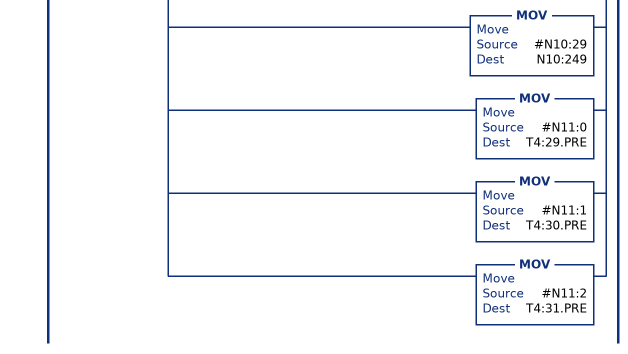
% Rung: 0 %
SOR SBR BST SUB N10:253 1 N10:254 NXB MUL N10:254 30 S:24 NXB MOV #N10:0 T4:0.PRE NXB MOV #N10:1 T4:1.PRE NXB MOV #N10:2 T4:2.PRE NXB MOV #N10:3 T4:3.PRE NXB MOV #N10:4 T4:4.PRE NXB MOV #N10:5 T4:5.PRE NXB MOV #N10:6 T4:6.PRE NXB MOV #N10:7 T4:7.PRE NXB MOV #N10:8 T4:8.PRE NXB MOV #N10:9 T4:9.PRE NXB MOV #N10:10 T4:11.PRE NXB MOV #N10:11 T4:12.PRE NXB MOV #N10:12 T4:13.PRE NXB MOV #N10:13 T4:15.PRE NXB MOV #N10:14 T4:18.PRE NXB MOV #N10:15 T4:19.PRE NXB MOV #N10:16 T4:20.PRE NXB MOV #N10:17 T4:21.PRE NXB MOV #N10:18 T4:22.PRE NXB MOV #N10:19 T4:25.PRE NXB MOV #N10:20 N10:240 NXB MOV #N10:21 N10:241 NXB MOV #N10:22 N10:242 NXB MOV #N10:23 N10:243 NXB MOV #N10:24 N10:244 NXB MOV #N10:25 N10:245 NXB MOV #N10:26 N10:246 NXB MOV #N10:27 N10:247 NXB MOV #N10:28 N10:248 NXB MOV #N10:29 N10:249 NXB MOV #N11:0 T4:29.PRE NXB MOV #N11:1 T4:30.PRE NXB MOV #N11:2 T4:31.PRE BND EOR
%   S:24  "Index Register" %

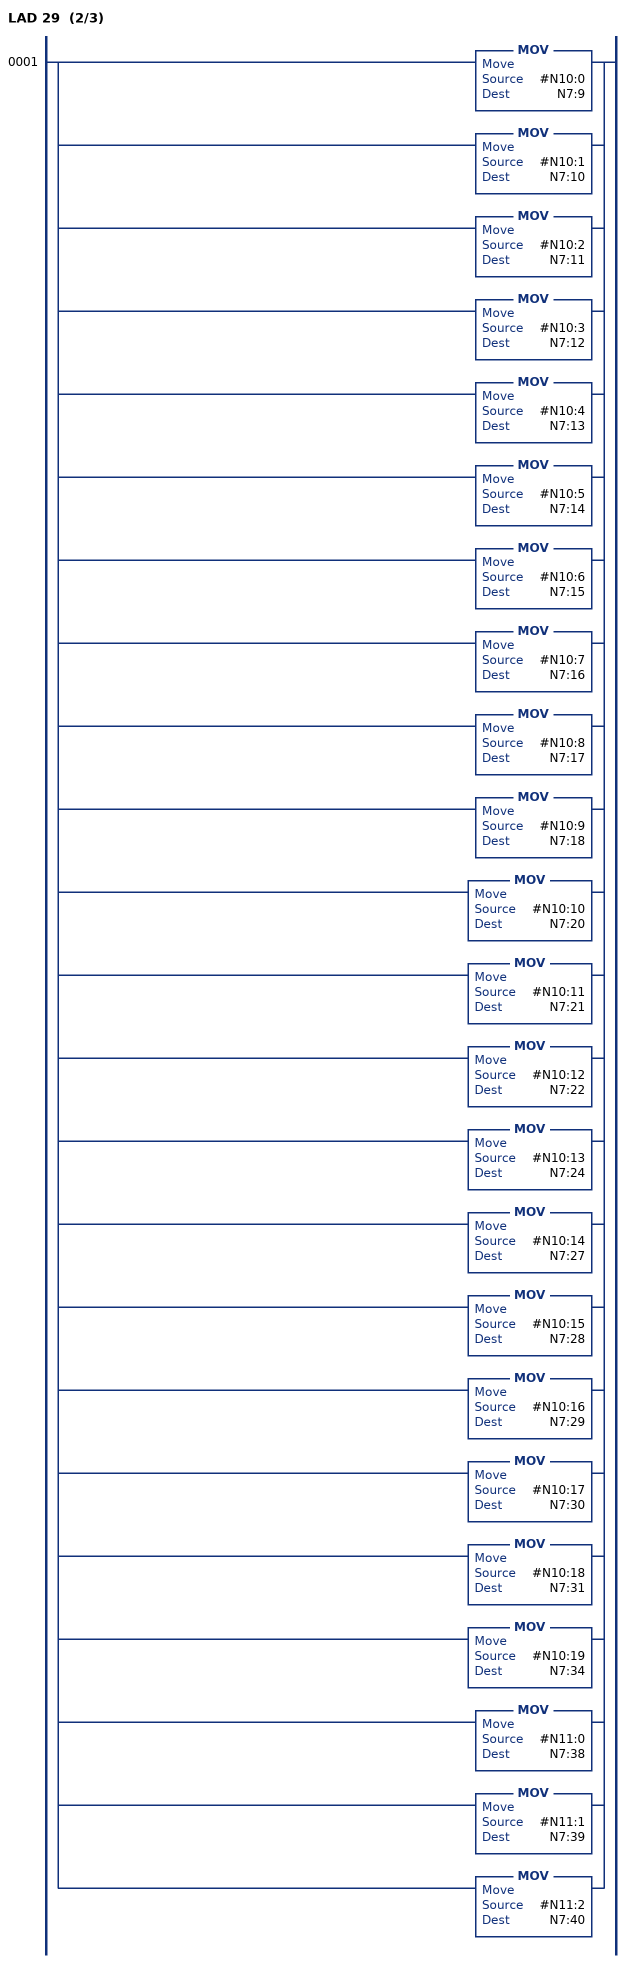
% Rung: 1 %
SOR BST MOV #N10:0 N7:9 NXB MOV #N10:1 N7:10 NXB MOV #N10:2 N7:11 NXB MOV #N10:3 N7:12 NXB MOV #N10:4 N7:13 NXB MOV #N10:5 N7:14 NXB MOV #N10:6 N7:15 NXB MOV #N10:7 N7:16 NXB MOV #N10:8 N7:17 NXB MOV #N10:9 N7:18 NXB MOV #N10:10 N7:20 NXB MOV #N10:11 N7:21 NXB MOV #N10:12 N7:22 NXB MOV #N10:13 N7:24 NXB MOV #N10:14 N7:27 NXB MOV #N10:15 N7:28 NXB MOV #N10:16 N7:29 NXB MOV #N10:17 N7:30 NXB MOV #N10:18 N7:31 NXB MOV #N10:19 N7:34 NXB MOV #N11:0 N7:38 NXB MOV #N11:1 N7:39 NXB MOV #N11:2 N7:40 BND EOR

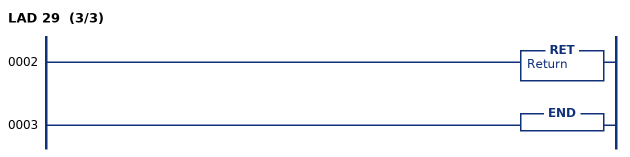
% Rung: 2 %
SOR RET EOR
% Rung: 3 %
SOR END EOR

LADDER 30
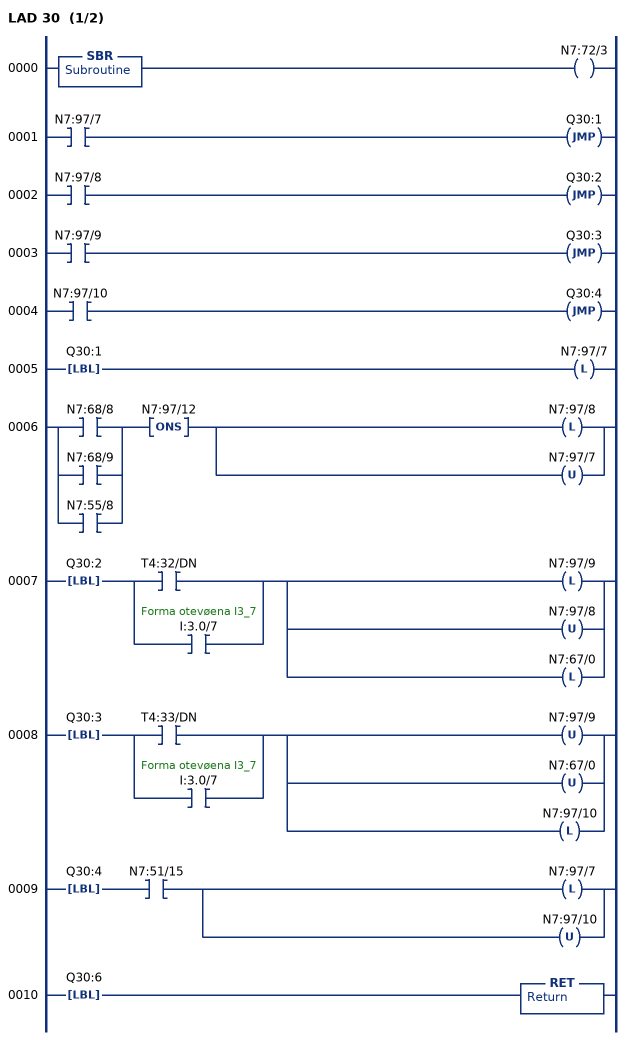
% Rung: 0 %
SOR SBR OTE N7:72/3 EOR
% Rung: 1 %
SOR XIC N7:97/7 JMP Q30:1 EOR
% Rung: 2 %
SOR XIC N7:97/8 JMP Q30:2 EOR
% Rung: 3 %
SOR XIC N7:97/9 JMP Q30:3 EOR
% Rung: 4 %
SOR XIC N7:97/10 JMP Q30:4 EOR
% Rung: 5 %
SOR LBL Q30:1 OTL N7:97/7 EOR
% Rung: 6 %
SOR BST XIC N7:68/8 NXB BST XIC N7:68/9 NXB XIC N7:55/8 BND BND OSR N7:97/12 BST OTL N7:97/8 NXB OTU N7:97/7 BND EOR
% Rung: 7 %
SOR LBL Q30:2 BST XIC T4:32/DN NXB XIC I:3.0/7 BND BST OTL N7:97/9 NXB BST OTU N7:97/8 NXB OTL N7:67/0 BND BND EOR
%   I:3.0/7  I3_7  "Forma otevøena" %
% Rung: 8 %
SOR LBL Q30:3 BST XIC T4:33/DN NXB XIC I:3.0/7 BND BST OTU N7:97/9 NXB BST OTU N7:67/0 NXB OTL N7:97/10 BND BND EOR
%   I:3.0/7  I3_7  "Forma otevøena" %
% Rung: 9 %
SOR LBL Q30:4 XIC N7:51/15 BST OTL N7:97/7 NXB OTU N7:97/10 BND EOR
% Rung: 10 %
SOR LBL Q30:6 RET EOR

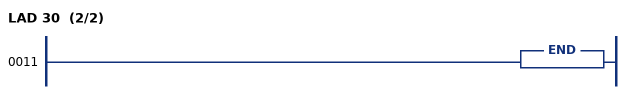
% Rung: 11 %
SOR END EOR

LADDER 31
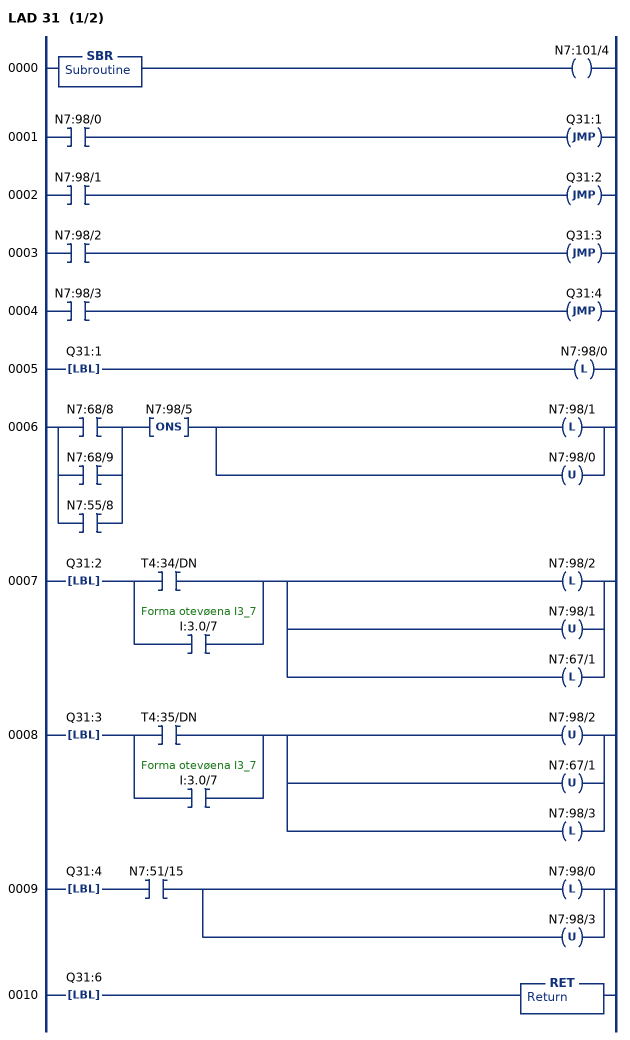
% Rung: 0 %
SOR SBR OTE N7:101/4 EOR
% Rung: 1 %
SOR XIC N7:98/0 JMP Q31:1 EOR
% Rung: 2 %
SOR XIC N7:98/1 JMP Q31:2 EOR
% Rung: 3 %
SOR XIC N7:98/2 JMP Q31:3 EOR
% Rung: 4 %
SOR XIC N7:98/3 JMP Q31:4 EOR
% Rung: 5 %
SOR LBL Q31:1 OTL N7:98/0 EOR
% Rung: 6 %
SOR BST XIC N7:68/8 NXB BST XIC N7:68/9 NXB XIC N7:55/8 BND BND OSR N7:98/5 BST OTL N7:98/1 NXB OTU N7:98/0 BND EOR
% Rung: 7 %
SOR LBL Q31:2 BST XIC T4:34/DN NXB XIC I:3.0/7 BND BST OTL N7:98/2 NXB BST OTU N7:98/1 NXB OTL N7:67/1 BND BND EOR
%   I:3.0/7  I3_7  "Forma otevøena" %
% Rung: 8 %
SOR LBL Q31:3 BST XIC T4:35/DN NXB XIC I:3.0/7 BND BST OTU N7:98/2 NXB BST OTU N7:67/1 NXB OTL N7:98/3 BND BND EOR
%   I:3.0/7  I3_7  "Forma otevøena" %
% Rung: 9 %
SOR LBL Q31:4 XIC N7:51/15 BST OTL N7:98/0 NXB OTU N7:98/3 BND EOR
% Rung: 10 %
SOR LBL Q31:6 RET EOR

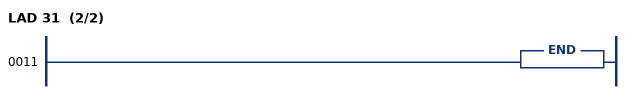
% Rung: 11 %
SOR END EOR

LADDER 32
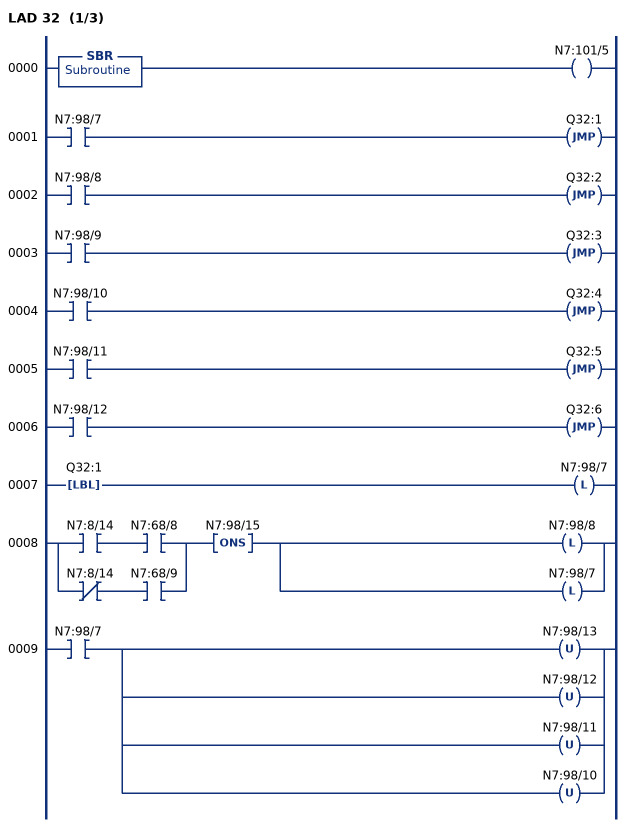
% Rung: 0 %
SOR SBR OTE N7:101/5 EOR
% Rung: 1 %
SOR XIC N7:98/7 JMP Q32:1 EOR
% Rung: 2 %
SOR XIC N7:98/8 JMP Q32:2 EOR
% Rung: 3 %
SOR XIC N7:98/9 JMP Q32:3 EOR
% Rung: 4 %
SOR XIC N7:98/10 JMP Q32:4 EOR
% Rung: 5 %
SOR XIC N7:98/11 JMP Q32:5 EOR
% Rung: 6 %
SOR XIC N7:98/12 JMP Q32:6 EOR
% Rung: 7 %
SOR LBL Q32:1 OTL N7:98/7 EOR
% Rung: 8 %
SOR BST XIC N7:8/14 XIC N7:68/8 NXB XIO N7:8/14 XIC N7:68/9 BND OSR N7:98/15 BST OTL N7:98/8 NXB OTL N7:98/7 BND EOR
% Rung: 9 %
SOR XIC N7:98/7 BST OTU N7:98/13 NXB BST OTU N7:98/12 NXB BST OTU N7:98/11 NXB OTU N7:98/10 BND BND BND EOR

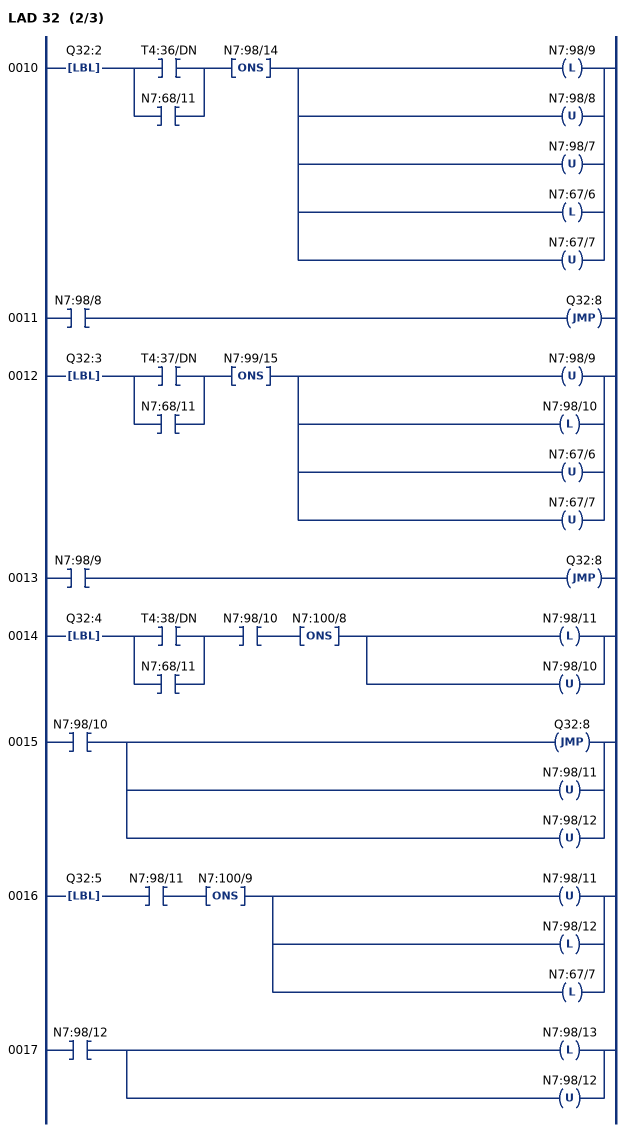
% Rung: 10 %
SOR LBL Q32:2 BST XIC T4:36/DN NXB XIC N7:68/11 BND OSR N7:98/14 BST OTL N7:98/9 NXB BST BST OTU N7:98/8 NXB OTU N7:98/7 BND NXB BST OTL N7:67/6 NXB OTU N7:67/7 BND BND BND EOR
% Rung: 11 %
SOR XIC N7:98/8 JMP Q32:8 EOR
% Rung: 12 %
SOR LBL Q32:3 BST XIC T4:37/DN NXB XIC N7:68/11 BND OSR N7:99/15 BST OTU N7:98/9 NXB BST OTL N7:98/10 NXB BST OTU N7:67/6 NXB OTU N7:67/7 BND BND BND EOR
% Rung: 13 %
SOR XIC N7:98/9 JMP Q32:8 EOR
% Rung: 14 %
SOR LBL Q32:4 BST XIC T4:38/DN NXB XIC N7:68/11 BND XIC N7:98/10 OSR N7:100/8 BST OTL N7:98/11 NXB OTU N7:98/10 BND EOR
% Rung: 15 %
SOR XIC N7:98/10 BST JMP Q32:8 NXB BST OTU N7:98/11 NXB OTU N7:98/12 BND BND EOR
% Rung: 16 %
SOR LBL Q32:5 XIC N7:98/11 OSR N7:100/9 BST BST OTU N7:98/11 NXB OTL N7:98/12 BND NXB OTL N7:67/7 BND EOR
% Rung: 17 %
SOR XIC N7:98/12 BST OTL N7:98/13 NXB OTU N7:98/12 BND EOR

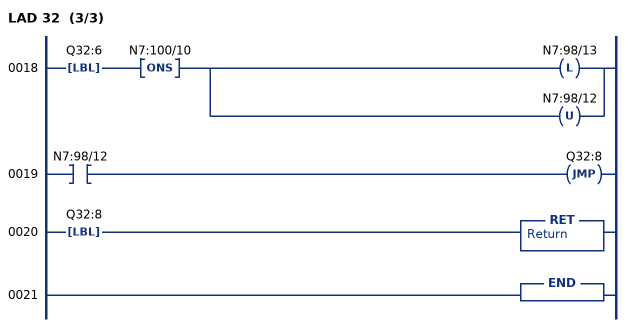
% Rung: 18 %
SOR LBL Q32:6 OSR N7:100/10 BST OTL N7:98/13 NXB OTU N7:98/12 BND EOR
% Rung: 19 %
SOR XIC N7:98/12 JMP Q32:8 EOR
% Rung: 20 %
SOR LBL Q32:8 RET EOR
% Rung: 21 %
SOR END EOR

LADDER 33
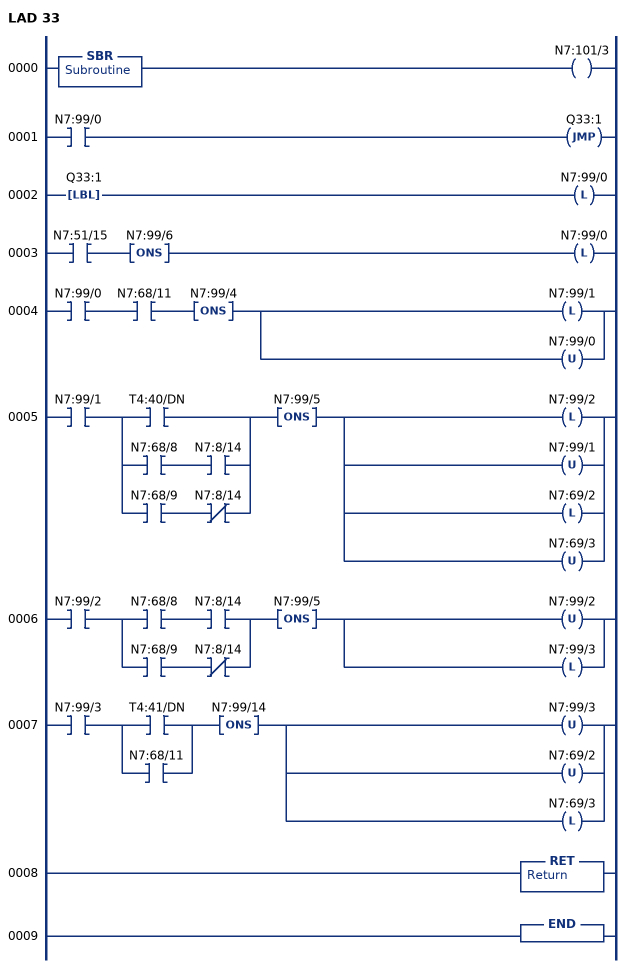
% Rung: 0 %
SOR SBR OTE N7:101/3 EOR
% Rung: 1 %
SOR XIC N7:99/0 JMP Q33:1 EOR
% Rung: 2 %
SOR LBL Q33:1 OTL N7:99/0 EOR
% Rung: 3 %
SOR XIC N7:51/15 OSR N7:99/6 OTL N7:99/0 EOR
% Rung: 4 %
SOR XIC N7:99/0 XIC N7:68/11 OSR N7:99/4 BST OTL N7:99/1 NXB OTU N7:99/0 BND EOR
% Rung: 5 %
SOR XIC N7:99/1 BST XIC T4:40/DN NXB BST XIC N7:68/8 XIC N7:8/14 NXB XIC N7:68/9 XIO N7:8/14 BND BND OSR N7:99/5 BST OTL N7:99/2 NXB BST OTU N7:99/1 NXB BST OTL N7:69/2 NXB OTU N7:69/3 BND BND BND EOR
% Rung: 6 %
SOR XIC N7:99/2 BST XIC N7:68/8 XIC N7:8/14 NXB XIC N7:68/9 XIO N7:8/14 BND OSR N7:99/5 BST OTU N7:99/2 NXB OTL N7:99/3 BND EOR
% Rung: 7 %
SOR XIC N7:99/3 BST XIC T4:41/DN NXB XIC N7:68/11 BND OSR N7:99/14 BST OTU N7:99/3 NXB BST OTU N7:69/2 NXB OTL N7:69/3 BND BND EOR
% Rung: 8 %
SOR RET EOR
% Rung: 9 %
SOR END EOR

LADDER 34
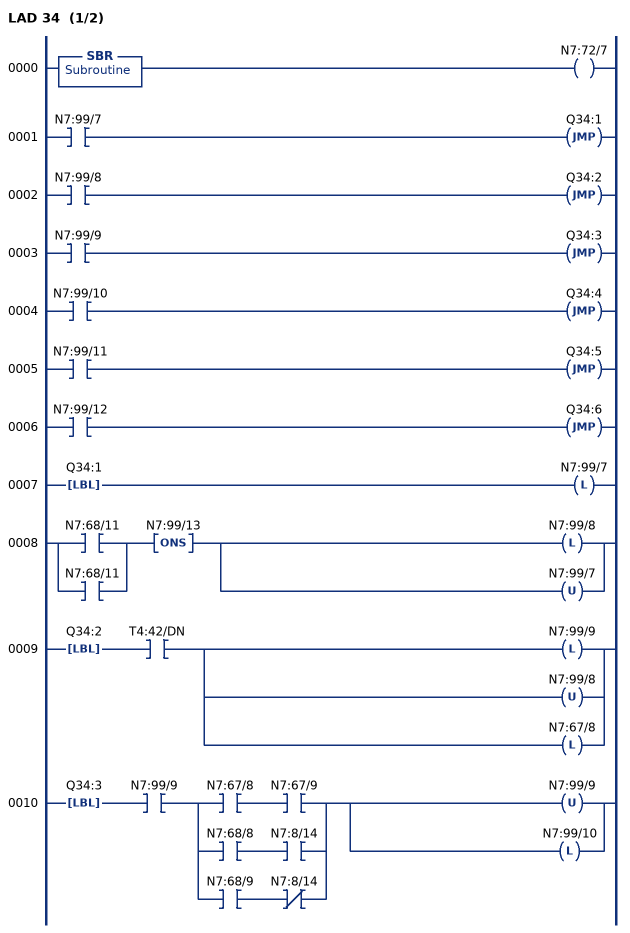
% Rung: 0 %
SOR SBR OTE N7:72/7 EOR
% Rung: 1 %
SOR XIC N7:99/7 JMP Q34:1 EOR
% Rung: 2 %
SOR XIC N7:99/8 JMP Q34:2 EOR
% Rung: 3 %
SOR XIC N7:99/9 JMP Q34:3 EOR
% Rung: 4 %
SOR XIC N7:99/10 JMP Q34:4 EOR
% Rung: 5 %
SOR XIC N7:99/11 JMP Q34:5 EOR
% Rung: 6 %
SOR XIC N7:99/12 JMP Q34:6 EOR
% Rung: 7 %
SOR LBL Q34:1 OTL N7:99/7 EOR
% Rung: 8 %
SOR BST XIC N7:68/11 NXB XIC N7:68/11 BND OSR N7:99/13 BST OTL N7:99/8 NXB OTU N7:99/7 BND EOR
% Rung: 9 %
SOR LBL Q34:2 XIC T4:42/DN BST OTL N7:99/9 NXB BST OTU N7:99/8 NXB OTL N7:67/8 BND BND EOR
% Rung: 10 %
SOR LBL Q34:3 XIC N7:99/9 BST XIC N7:67/8 XIC N7:67/9 NXB BST XIC N7:68/8 XIC N7:8/14 NXB XIC N7:68/9 XIO N7:8/14 BND BND BST OTU N7:99/9 NXB OTL N7:99/10 BND EOR

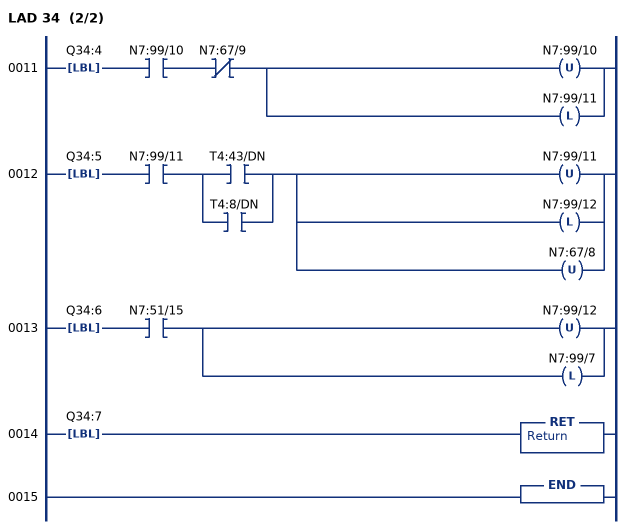
% Rung: 11 %
SOR LBL Q34:4 XIC N7:99/10 XIO N7:67/9 BST OTU N7:99/10 NXB OTL N7:99/11 BND EOR
% Rung: 12 %
SOR LBL Q34:5 XIC N7:99/11 BST XIC T4:43/DN NXB XIC T4:8/DN BND BST OTU N7:99/11 NXB BST OTL N7:99/12 NXB OTU N7:67/8 BND BND EOR
% Rung: 13 %
SOR LBL Q34:6 XIC N7:51/15 BST OTU N7:99/12 NXB OTL N7:99/7 BND EOR
% Rung: 14 %
SOR LBL Q34:7 RET EOR
% Rung: 15 %
SOR END EOR

LADDER 35
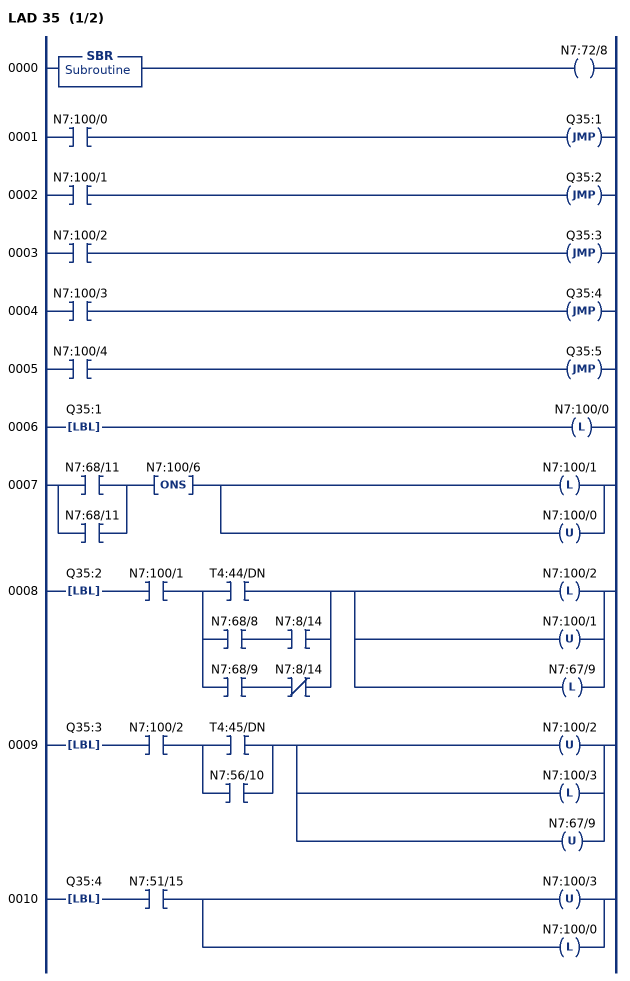
% Rung: 0 %
SOR SBR OTE N7:72/8 EOR
% Rung: 1 %
SOR XIC N7:100/0 JMP Q35:1 EOR
% Rung: 2 %
SOR XIC N7:100/1 JMP Q35:2 EOR
% Rung: 3 %
SOR XIC N7:100/2 JMP Q35:3 EOR
% Rung: 4 %
SOR XIC N7:100/3 JMP Q35:4 EOR
% Rung: 5 %
SOR XIC N7:100/4 JMP Q35:5 EOR
% Rung: 6 %
SOR LBL Q35:1 OTL N7:100/0 EOR
% Rung: 7 %
SOR BST XIC N7:68/11 NXB XIC N7:68/11 BND OSR N7:100/6 BST OTL N7:100/1 NXB OTU N7:100/0 BND EOR
% Rung: 8 %
SOR LBL Q35:2 XIC N7:100/1 BST XIC T4:44/DN NXB BST XIC N7:68/8 XIC N7:8/14 NXB XIC N7:68/9 XIO N7:8/14 BND BND BST OTL N7:100/2 NXB BST OTU N7:100/1 NXB OTL N7:67/9 BND BND EOR
% Rung: 9 %
SOR LBL Q35:3 XIC N7:100/2 BST XIC T4:45/DN NXB XIC N7:56/10 BND BST OTU N7:100/2 NXB BST OTL N7:100/3 NXB OTU N7:67/9 BND BND EOR
% Rung: 10 %
SOR LBL Q35:4 XIC N7:51/15 BST OTU N7:100/3 NXB OTL N7:100/0 BND EOR

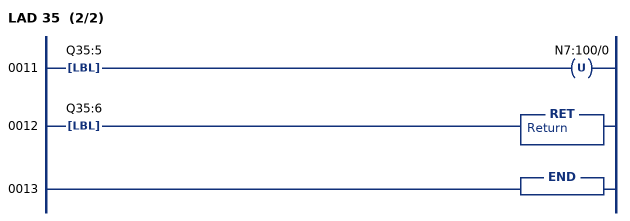
% Rung: 11 %
SOR LBL Q35:5 OTU N7:100/0 EOR
% Rung: 12 %
SOR LBL Q35:6 RET EOR
% Rung: 13 %
SOR END EOR

OTHER DOCUMENTED ADDRESSES
  I:1.0/2  I1_2  "Chlazení oleje"
  I:1.0/6  I1_6  "Akumulátor není vypouštìn"
  I:2.0/1  I2_1  "Rezerva 2"
  I:2.0/2  I2_2  "Rezerva 3"
  I:9.1  I9_1_WORD  "Otáèky šneku vytlaè. stroje"
  O:5.0/15  O5_15  "Chlazení formy vodou _|"
  O:8.0/13  O8_13

SYMBOL GROUPS
  VSTUPY: I:1.0/15 I:9.1 I:9.0 I:2.0/15 I:2.0/14 I:1.0/0 I:1.0/2 I:1.0/1 I:1.0/3 I:1.0/4 I:1.0/5 I:1.0/6 I:1.0/7 I:1.0/8 I:1.0/9 I:1.0/10 I:1.0/11 I:1.0/12 I:1.0/13 I:1.0/14 I:2.0/0 I:2.0/1 I:2.0/2 I:2.0/3 I:2.0/4 I:2.0/5 I:2.0/6 I:2.0/7 I:2.0/8 I:2.0/9 I:2.0/10 I:2.0/11 I:2.0/12 I:2.0/13 I:3.0/0 I:3.0/1 I:3.0/2 I:3.0/3 I:3.0/4 I:3.0/5 I:3.0/6 I:3.0/7 I:3.0/8 I:3.0/9 I:3.0/10 I:3.0/11 I:3.0/12 I:3.0/13 I:3.0/14 I:3.0/15 I:4.0/0 I:4.0/1 I:4.0/2 I:4.0/3 I:4.0/4 I:4.0/5 I:4.0/6 I:4.0/7 I:4.0/8 I:4.0/9 I:4.0/10 I:4.0/11 I:4.0/12 I:4.0/13 I:4.0/14 I:4.0/15
  VÝSTUPY: O:5.0/0 O:5.0/1 O:5.0/2 O:5.0/3 O:5.0/4 O:5.0/5 O:5.0/6 O:5.0/7 O:5.0/8 O:5.0/9 O:5.0/10 O:5.0/11 O:5.0/12 O:5.0/13 O:5.0/14 O:5.0/15 O:6.0/0 O:6.0/1 O:6.0/2 O:6.0/3 O:6.0/4 O:6.0/5 O:6.0/6 O:6.0/7 O:6.0/8 O:6.0/9 O:6.0/10 O:6.0/11 O:6.0/12 O:6.0/13 O:6.0/14 O:6.0/15 O:7.0/0 O:7.0/1 O:7.0/2 O:7.0/3 O:7.0/4 O:7.0/5 O:7.0/6 O:7.0/7 O:7.0/8 O:7.0/9 O:7.0/10 O:7.0/11 O:7.0/12 O:7.0/13 O:7.0/14 O:7.0/15 O:8.0/0 O:8.0/1 O:8.0/2 O:8.0/3 O:8.0/4 O:8.0/5 O:8.0/6 O:8.0/7 O:8.0/8 O:8.0/9 O:8.0/10 O:8.0/11 O:8.0/12 O:8.0/13 O:8.0/14 O:8.0/15

DATA TABLE (non-zero values as saved)
DATA T4
% .PRE .ACC %
% T4:0 % 3600 0
% T4:1 % 3800 0
% T4:2 % 3500 0
% T4:3 % 35 0
% T4:4 % 1000 0
% T4:5 % 118 0
% T4:6 % 60 0
% T4:7 % 3050 0
% T4:8 % 680 0
% T4:9 % 80 0
% T4:10 % 400 0
% T4:11 % 5 0
% T4:12 % 20 0
% T4:13 % 300 0
% T4:14 % 400 0
% T4:15 % 60 0
% T4:16 % 40 5
% T4:17 % 40 0
% T4:23 % 2000 0
% T4:24 % 500 0
% T4:25 % 10 0
% T4:26 % 2000 0
% T4:27 % 50 50
% T4:28 % 500 0
% T4:29 % 0 1
% T4:31 % 0 1
% T4:32 % 40 0
% T4:33 % 500 0
% T4:34 % 50 0
% T4:35 % 500 0
% T4:36 % 50 0
% T4:37 % 100 0
% T4:39 % 50 50
% T4:40 % 71 0
% T4:46 % 750 0
% T4:47 % 1 0
% T4:48 % 100 0
% T4:49 % 1800 0
% T4:50 % 10 0
DATA C5
% .PRE .ACC %
% C5:0 % 30000 3742
% C5:1 % 0 31359
% C5:2 % 30000 0
% C5:3 % 10 0
% C5:4 % 1000 38
DATA N7
% N7:0 % 0 0 0 0 0 0 0 0 256 3600
% N7:10 % 3800 3500 35 1000 118 60 3050 680 80 200
% N7:20 % 5 20 300 300 60 40 40 0 0 0
% N7:30 % 0 0 1700 500 10 500 50 400 0 0
% N7:40 % 0 0 0 0 -32640 0 0 0 1 0
% N7:50 % 4108 32 0 0 0 4096 1 16385 256 64
% N7:60 % 0 -32768 0 0 64 0 0 0 0 0
% N7:70 % 2992 1 0 0 0 0 16387 40 500 50
% N7:80 % 500 50 100 0 50 71 0 0 0 0
% N7:90 % 0 750 0 0 0 1 0 1153 0 0
% N7:100 % 8192 1 100 1800 10 0 0 0 0 0
DATA N10
% N10:0 % 5000 500 4300 200 4000 200 20 4500 400 20
% N10:10 % 200 20 20 150 300 50 200 400 600 800
% N10:30 % 1500 1500 1350 100 900 350 20 1300 100 100
% N10:40 % 200 20 20 150 300 50 0 200 750 950
% N10:50 % 1800 1850 1900 1900 1900 1900 1850 1850 0 380
% N10:60 % 1500 1500 1350 200 900 350 20 1300 100 20
% N10:70 % 200 20 20 110 300 50 200 400 600 800
% N10:90 % 1500 500 100 300 900 200 20 1300 150 20
% N10:100 % 200 20 20 150 300 50 200 400 600 800
% N10:120 % 1500 500 100 300 900 200 20 1300 150 20
% N10:130 % 200 20 20 150 300 50 200 400 600 800
% N10:150 % 1500 500 100 300 900 200 20 1300 150 20
% N10:160 % 200 20 20 150 300 50 200 400 600 800
% N10:180 % 1500 500 100 300 900 200 20 1300 150 20
% N10:190 % 200 20 20 150 300 50 200 400 600 800
% N10:210 % 1500 500 100 300 900 200 20 1300 150 20
% N10:220 % 200 20 20 150 300 50 200 400 600 800
% N10:250 % 2 2 1 2 1 16384
